{attribute 'qualified_only'}
{attribute addProperty Name "IO"}
VAR_GLOBAL
    {attribute addProperty Name "A1"}
    A1 : InputsBase_8;
    {attribute addProperty Name "A2"}
    A2 : OutputsBase_8;
    {attribute addProperty Name "A3"}
    A3 : AnalogInputsBase_4;
    {attribute addProperty Name "A4"}
    A4 : AnalogOutputsBase_4;
END_VAR

(* stored: Version 1.1.0.1, ProductVersion 3.1.4024.9
   GVL IO: Id {8542ff68-7604-0fca-1820-2083dd0a2bfb} *)
